{attribute 'linkalways'} 
{attribute 'no_explicit_call' := 'This FB is a CLASS and must be accessed using methods or properties'}
{attribute 'enable_dynamic_creation'}
FUNCTION_BLOCK FINAL NOT_DWORD EXTENDS Node
VAR
	in : _DWORD(0);
	out : _DWORD(0);
END_VAR

METHOD PUBLIC Clone : I_Node
VAR
	pNode : POINTER TO NOT_DWORD;
END_VAR
pNode := __NEW(NOT_DWORD);
Clone := pNode^;
END_METHOD

METHOD FB_init : BOOL
VAR_INPUT
	bInitRetains : BOOL; // if TRUE, the retain variables are initialized (warm start / cold start)
	bInCopyCode : BOOL;  // if TRUE, the instance afterwards gets moved into the copy code (online change)
END_VAR
AddInput('in',THIS^.in);
AddOutput('out', THIS^.out);
END_METHOD

METHOD PROTECTED OnExecute
VAR
END_VAR
out.Value := NOT in.Value;
END_METHOD

END_FUNCTION_BLOCK

(* stored: Version 1.1.0.1, ProductVersion 3.1.4024.15
   POU NOT_DWORD: Id {67f75d2e-cdc1-42cb-b0bd-8520061e05fe}, SpecialFunc None
   Folder Constructor: Id {a604b36c-bd8f-46f9-addd-41861d6d8f79}
   Method Clone: Id {d981be77-107f-4191-a67b-79b78ad84534}
   Method FB_init: Id {b306f46b-f561-4f2d-b99f-c99288d2cc38}
   Method OnExecute: Id {b37ec9f3-a70e-4095-bfe6-715da60e9b78} *)
